{attribute 'qualified_only'}
{attribute 'strict'}
TYPE eMotorStates :
(
	firstrun, running, stopped, errored, starting, stopping, pause, paused
);
END_TYPE

(* stored: Version 1.1.0.1, ProductVersion 3.1.4024.12
   DUT eMotorStates: Id {e6434275-2629-4ba6-addb-744d5ee1f572} *)
